// TIA Portal V20 export
TYPE "LConSMC_typeSectionalDriveTorquePrecontrolConfig"
// Konfigurationsdaten der Momentenvorsteuerung einer Bahnzugregelung / Configuration data of torque precontrol for sectional drives
// stored: Access Published
   STRUCT
      useSetValForFrictionComp : Bool := FALSE;   // TRUE: Drehzahl-Sollwert wird für die Kompensastion der Reibung verwendet FALSE: Drehzahl-Istwert wird für die Kompensation der Reibung verwendet / TRUE: Use speed setpoint for friction compensation FALSE: Use speed actual value
      frictionAdjustment : Real := 0.0;   // Multiplikativer Faktor zur Adaption des Reibmomentes (1.0 = 100%) / Multiplicative adaption factor for friction torque (1.0 = 100%)
      xn_speedValues { S7_SetPoint := 'True'} : "LConSMC_typeBreakPointTable";   // [1/min] Drehzahlwerte der Reibkennlinie / [1/min] Speed values for fiction characteristic
      yn_torqueValues { S7_SetPoint := 'True'} : "LConSMC_typeBreakPointTable";   // [Nm oder lbf ft] Drehmomentenwerte der Reibkennlinie / [Nm or lbf ft] Torque values for friction characteristic
      sizeOfArray : Int := 20;   // Anzahl verwendeter Stützpunkte der Reibkennlinie / Size of friction characteristic array
      loadGear { S7_SetPoint := 'True'} : "LConSMC_typeLoadGear";   // Motorgetriebe / Load gear settings
      JFixed : LReal;   // [kgm^2] / [lbft^2] Trägheit bezogen auf Motorseite (ohne Motor, z.B. Getriebe) / [kgm^2] / [lbft^2] Inertia on drive side (without drive, e.g. gear box)
      JMandrel : LReal;   // [kgm^2] / [lbft^2] Trägheit auf der Lastseite (z.B. Rolle) / [kgm^2] / [lbft^2] Inertia on load side (e.g. mandrel)
      JMotor : LReal;   // [kgm^2] / [lbft^2] Motorträgheit / [kgm^2] / [lbft^2] Drive inertia
      tensionAdjustment : Real := 0.0;   // Multiplikativer Faktor zur Adaption des Zugmomentes (1.0 = 100%) / Multiplicative adaption factor for tension torque (1.0 = 100%)
      accelerationAdjustment : Real := 1.0;   // Multiplikativer Faktor zur Adaption des Beschleunigungsmomentes aus der Bahnbeschleunigung (1.0 = 100%) / Multiplicative adaption factor for acceleration torque from web acceleration (1.0 = 100%)
      upperTorqueLimit : LReal := 1.0;   // [%] 1.0 = 100% Obere Drehmomentengrenze 0-200% des Bezugsmomentes / [%] 1.0 = 100% Upper torque limit 0..200% of nominal torque
      lowerTorqueLimit : LReal := -1.0;   // [%] 1.0 = 100% Untere Drehmomentengrenze 0-200% des Bezugsmomentes / [%] 1.0 = 100% Lower torque limit (0..-200% of nominal torque)
      referenceTorque : LReal;   // Referenzdrehmoment (SINAMICS p2003) !Nur notwendig wenn "getAxisConfigAtStart" = FALSE! / Reference torque (SINAMICS p2003) !Only necessary if "getAxisConfigAtStart" = FALSE!
   END_STRUCT;
   // xn_speedValues.values[0..19] := 0.0;
   // yn_torqueValues.values[0..19] := 0.0;
END_TYPE
